FUNCTION FC_PRG1 : BOOL
VAR_INPUT
END_VAR
VAR

	Stap : DINT;
	
END_VAR


CASE Stap OF
	
	
	
	
END_CASE

END_FUNCTION

(* stored: Version 1.1.0.1, ProductVersion 3.1.4024.12
   POU FC_PRG1: Id {3c2d693e-a12f-40bc-9ef3-094978264baf}, SpecialFunc None *)
